// SIMATIC S7-200 project (STEP 7-Micro/WIN), CPU 221 REL 01.10

SYMBOL_TABLE USER1
bezczynnosc_do_za_gorac M1.7     // w彻cz wiatrak
bezczynnosc_do_za_zimno M1.6     // w彻cz grzanie
ANDwb            M1.5     // wy彻czenie wiatraka
ANDgb            M1.4     // wy彻czenie grza砶i
RSwentylator     M1.3
RSgrzalka        M1.2
RSbezczynnosc    M1.1
ANDgrzalka       M0.6
bezczynnosc      M0.5
ANDwentylator    M0.7
T_z_sub_h        VW130
T_z_add_h        VW120
h                VW110
T_ge_T_z         M0.2
T_z_ge_T         M0.1
h_count          C1
T_z              VW100
T_z_count        C0
T                AIW8
END_SYMBOL_TABLE

ORGANIZATION_BLOCK MAIN:OB1
TITLE=PROGRAM COMMENTS
BEGIN
Network 1
// AND wentylator  (dodac T> T_z + h)
// (network saved uncompiled; FBD cells follow)
// row 1: c2 [AND ?0_20_0 RSbezczynnosc:M1.1 ANDwentylator:M0.7 ]
// row 2: c2 [box]
// row 3: c2 [box]
Network 2
// AND grzalka (dodac T_z - h > T)
// (network saved uncompiled; FBD cells follow)
// row 1: c2 [AND ?0_20_0 RSbezczynnosc:M1.1 ANDgrzalka:M0.6 ]
// row 2: c2 [box]
// row 3: c2 [box]
Network 3
// AND grzalka -> bezczynnosc (dodac T >= T_z)
// (network saved uncompiled; FBD cells follow)
// row 1: c2 [AND ?0_20_0 RSgrzalka:M1.2 ANDgb:M1.4 ]
// row 2: c2 [box]
// row 3: c2 [box]
Network 4
// AND wentylator -> bezczynnosc (dodac T <= T_z)
// (network saved uncompiled; FBD cells follow)
// row 2: c2 [AND ?0_20_0 RSwentylator:M1.3 ANDwb:M1.5 ]
// row 3: c2 [box]
// row 4: c2 [box]
Network 5
// (network saved uncompiled; FBD cells follow)
// row 1: c1 [OR SM0.1 ANDgb:M1.4 ANDwb:M1.5 ]  c2 --  c3 [RS Q0.3 S:=power@row1, R1:=power@row5, OUT=>power]  c4 --  c5 -- v  c6 --  c7 --  c8 [= RSbezczynnosc:M1.1 ]
// row 2: c1 [box]  c3 [box]  c5 ^v
// row 3: c1 [box]  c3 [box]  c5 ^  c6 --  c7 [= V0.0 ]
// row 4: c1 [box]  c3 [box]
// row 5: c1 [OR ANDwentylator:M0.7 ANDgrzalka:M0.6 ]  c2 --  c3 [box]
// row 6: c1 [box]
Network 6
// w彻cz wiatrak
// (network saved uncompiled; FBD cells follow)
// row 1: c1 [RS Q0.1 S:=ANDwentylator:M0.7, R1:=ANDwb:M1.5, OUT=>power]  c2 -- v  c3 --  c4 [= RSwentylator:M1.3 ]
// row 2: c1 [box]  c2 ^v
// row 3: c2 ^  c3 --  c4 [= V0.0 ]
Network 7
// w彻cz grzanie
// (network saved uncompiled; FBD cells follow)
// row 1: c1 [RS Q0.2 S:=ANDgrzalka:M0.6, R1:=ANDgb:M1.4, OUT=>power]  c2 -- v  c3 --  c4 --  c5 [= RSgrzalka:M1.2 ]
// row 2: c1 [box]  c2 ^v
// row 3: c1 [box]  c2 ^  c3 --  c4 [= V0.0 ]
END_ORGANIZATION_BLOCK
